FUNCTION_BLOCK PnPSensor (* Proximity sensor detect the presence of object at a specific position *)
  (* Standard: 61499-2 *)
  (* Version 1.0, 2008-11-09, Cheng Pang, The University of Auckland, Stable build. *)
  (* Compiler header: package fb.rt.pnp; *)
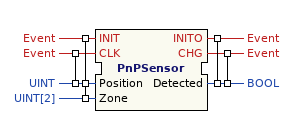
  EVENT_INPUT
    INIT WITH Position, Zone; (* Initialization Request *)
    CLK WITH Position; (* Clock signal *)
  END_EVENT
  EVENT_OUTPUT
    INITO WITH Detected; (* Initialization Confirm *)
    CHG WITH Detected; (* Value of DETECTED changed *)
  END_EVENT
  VAR_INPUT
    Position : UINT; (* The object's position *)
    Zone : ARRAY [0..1] OF UINT; (* Detection range of the sensor *)
  END_VAR
  VAR_OUTPUT
    Detected : BOOL; (* Whether an object is detected *)
  END_VAR
  VAR
    emitCHG : BOOL;
  END_VAR
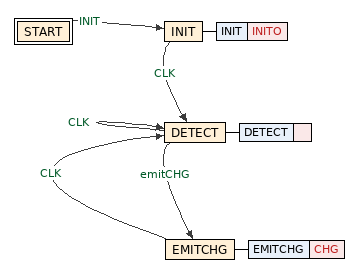
  EC_STATES
    START; (* Initial State *)
    INIT : INIT -> INITO; (* Initialization *)
    DETECT : DETECT; (* Detect *)
    EMITCHG : EMITCHG -> CHG;
  END_STATES
  EC_TRANSITIONS
    START TO INIT := INIT;
    INIT TO DETECT := CLK;
    DETECT TO DETECT := CLK;
    DETECT TO EMITCHG := emitCHG;
    EMITCHG TO DETECT := CLK;
  END_TRANSITIONS
  ALGORITHM INIT IN Java: (* Initialization algorithm *)
if((Position.value>=((UINT)Zone.value[0]).value)&&(Position.value<=((UINT)Zone.value[1]).value)){
  Detected.value = true;
}
else{
  Detected.value = false;
}
emitCHG.value = false;
  END_ALGORITHM
  ALGORITHM DETECT IN Java: (* Normally executed algorithm *)
if((Position.value>=((UINT)Zone.value[0]).value)&&(Position.value<=((UINT)Zone.value[1]).value)){
  if(Detected.value==false){
    Detected.value = true;
    emitCHG.value = true;
  }
}
else{
  if(Detected.value==true){
    Detected.value = false;
    emitCHG.value = true;
  }
}
  END_ALGORITHM
  ALGORITHM EMITCHG IN ST:
emitCHG := FALSE;
  END_ALGORITHM
END_FUNCTION_BLOCK
